FUNCTION_BLOCK Selector (* Extracted Composite Function Block Type *)
  (* Standard: 61499-2 *)
  (* Version 2/18/2024, midxav *)
  PACKAGE Main;
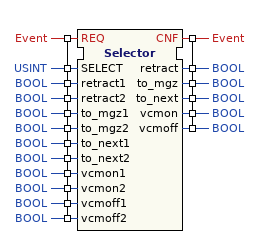
  EVENT_INPUT
    REQ WITH SELECT, retract1, retract2, to_mgz1, to_mgz2, to_next1, to_next2, vcmon1, vcmon2, vcmoff1, vcmoff2; (* Normal Execution Request *)
  END_EVENT
  EVENT_OUTPUT
    CNF WITH retract, to_mgz, to_next, vcmon, vcmoff; (* Execution Confirmation *)
  END_EVENT
  VAR_INPUT
    SELECT : USINT; (* Selector *)
    retract1 : BOOL;
    retract2 : BOOL;
    to_mgz1 : BOOL;
    to_mgz2 : BOOL;
    to_next1 : BOOL;
    to_next2 : BOOL;
    vcmon1 : BOOL;
    vcmon2 : BOOL;
    vcmoff1 : BOOL;
    vcmoff2 : BOOL;
  END_VAR
  VAR_OUTPUT
    retract : BOOL;
    to_mgz : BOOL;
    to_next : BOOL;
    vcmon : BOOL;
    vcmoff : BOOL;
  END_VAR
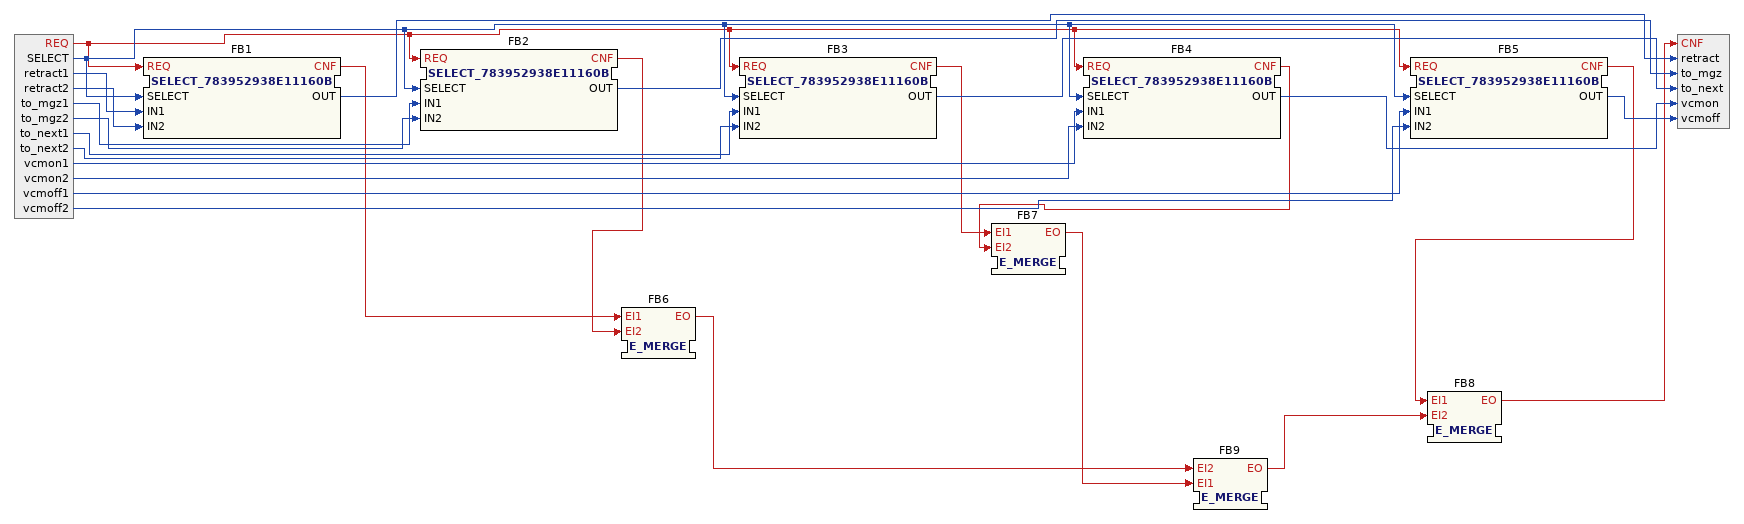
  FBS
    FB1 : SELECT_783952938E11160B; {SET_ATTRIBUTE(Configuration.GenericFBType.InterfaceParams, Runtime.Standard#CNT:=2;IN${CNT$}:BOOL)}
    FB2 : SELECT_783952938E11160B; {SET_ATTRIBUTE(Configuration.GenericFBType.InterfaceParams, Runtime.Standard#CNT:=2;IN${CNT$}:BOOL)}
    FB3 : SELECT_783952938E11160B; {SET_ATTRIBUTE(Configuration.GenericFBType.InterfaceParams, Runtime.Standard#CNT:=2;IN${CNT$}:BOOL)}
    FB4 : SELECT_783952938E11160B; {SET_ATTRIBUTE(Configuration.GenericFBType.InterfaceParams, Runtime.Standard#CNT:=2;IN${CNT$}:BOOL)}
    FB5 : SELECT_783952938E11160B; {SET_ATTRIBUTE(Configuration.GenericFBType.InterfaceParams, Runtime.Standard#CNT:=2;IN${CNT$}:BOOL)}
    FB6 : E_MERGE;
    FB7 : E_MERGE;
    FB8 : E_MERGE;
    FB9 : E_MERGE;
  END_FBS
  EVENT_CONNECTIONS
    REQ TO FB1.REQ;
    REQ TO FB2.REQ;
    REQ TO FB3.REQ;
    REQ TO FB4.REQ;
    REQ TO FB5.REQ;
    FB1.CNF TO FB6.EI1;
    FB2.CNF TO FB6.EI2;
    FB3.CNF TO FB7.EI1;
    FB4.CNF TO FB7.EI2;
    FB5.CNF TO FB8.EI1;
    FB6.EO TO FB9.EI2;
    FB7.EO TO FB9.EI1;
    FB9.EO TO FB8.EI2;
    FB8.EO TO CNF;
  END_CONNECTIONS
  DATA_CONNECTIONS
    SELECT TO FB1.SELECT;
    SELECT TO FB2.SELECT;
    SELECT TO FB3.SELECT;
    SELECT TO FB4.SELECT;
    SELECT TO FB5.SELECT;
    FB1.OUT TO retract;
    FB2.OUT TO to_mgz;
    FB3.OUT TO to_next;
    FB4.OUT TO vcmon;
    FB5.OUT TO vcmoff;
    retract1 TO FB1.IN1;
    retract2 TO FB1.IN2;
    to_mgz1 TO FB2.IN1;
    to_mgz2 TO FB2.IN2;
    to_next1 TO FB3.IN1;
    to_next2 TO FB3.IN2;
    vcmon1 TO FB4.IN1;
    vcmon2 TO FB4.IN2;
    vcmoff1 TO FB5.IN1;
    vcmoff2 TO FB5.IN2;
  END_CONNECTIONS
END_FUNCTION_BLOCK
